FUNCTION UpdateEventTimeStampSystemTime
VAR_INPUT
	stEvent : REFERENCE TO ST_Event;
END_VAR
VAR
	fbGETSYSTEMTIME : GETSYSTEMTIME;
	stFileTime : T_FILETIME;
END_VAR

fbGETSYSTEMTIME (TimeLoDW => stFileTime.dwLowDateTime,
				TimeHiDW => stFileTime.dwHighDateTime);

stEvent.dtTimeStamp := FILETIME_TO_DT (fileTime := stFileTime);

END_FUNCTION

(* stored: Version 1.1.0.1, ProductVersion 3.1.4024.12
   POU UpdateEventTimeStampSystemTime: Id {87bbf23c-4db1-48e1-9623-b2b331c9a59b}, SpecialFunc None *)
